TEXTLIST GLP_Available
  0 = 'Not Available'
  1 = 'Available'
   = ''
END_TEXTLIST

(* stored: Version 1.1.0.1, ProductVersion 3.1.4024.12
   TextList GLP_Available: Id {b7c2a945-f444-4152-bc31-9c3de09a0d87} *)
